FUNCTION_BLOCK FB_StateMaint
VAR_IN_OUT
	stAxis  	: ARRAY [GVL.cXP .. GVL.cXM] OF ST_AxisGroup;
	bTopEntry	: BOOL;
END_VAR
VAR_INPUT
	eCommand			: E_Commands;
	stCalibrate			: ST_Calibrate;
	stChangeAxisEnable	: ST_ChangeAxisEnable;
	stChangeBrakeState	: ST_ChangeBrakeState;
	stClearAllFaults	: ST_ClearAllFaults;
	stClearAxisFaults	: ST_ClearAxisFaults;
	stDisableAllAxes	: ST_DisableAllAxes;
	stEnableAllAxes		: ST_EnableAllAxes;
	stGoToProd			: ST_GoToProd;
	stHomeAxis			: ST_HomeAxis;
	stMoveAxisAbsolute	: ST_MoveAxisAbsolute;
	stMoveAxisRelative	: ST_MoveAxisRelative;
END_VAR
VAR_OUTPUT
	bCalibDone		: BOOL;
	bMotionDone		: BOOL;
	stOutCalibDone	: ST_CalibDone;
	nSMState		: DINT;
END_VAR
VAR
	//state-machine
	eCurrentState	: E_StatesMaint;
	eNextState		: E_StatesMaint;
	fbHoming		: FB_Homing;
	fbCalibrating	: FB_StateCalibrating;
	fbMoving		: FB_StateMoving;
	fbStill			: FB_StateStill;
	bLowerEntry 	: BOOL;

	//other var
	eCopyCommand	: E_Commands;
	fbCalibRtrig	: R_TRIG;
	bCalibRestart : BOOL;
	
	//testVar
	a, b, c : INT;
	
END_VAR


IF bTopEntry = TRUE THEN
	bTopEntry := FALSE;
	eNextState := E_StatesMaint.Still;
END_IF	
IF eCurrentState <> eNextState THEN
	bLowerEntry := TRUE;
END_IF
eCurrentState := eNextState;
nSMState := eCurrentState;
bMotionDone := FALSE;
//State Machine
CASE eCurrentState OF
	
	E_StatesMaint.Still:
		bCalibRestart := TRUE;
		fbStill(
			stAxis				:= stAxis, 
			bTopEntry			:= bLowerEntry, 
			eCommand			:= eCommand,
			stChangeAxisEnable 	:= stChangeAxisEnable,
			stChangeBrakeState	:= stChangeBrakeState,
			stClearAllFaults	:= stClearAllFaults,
			stClearAxisFaults	:= stClearAxisFaults,
			stDisableAllAxes	:= stDisableAllAxes,
			stEnableAllAxes		:= stEnableAllAxes);
		IF eCommand <> E_Commands.noCommand THEN (*checks if there is a new command*)
			IF eCommand = E_Commands.calibrate THEN
				eNextState := E_StatesMaint.Calibrating;
			ELSIF eCommand = E_Commands.closeShutter OR_ELSE
				eCommand = E_Commands.homeAxis OR_ELSE
				eCommand = E_Commands.moveAxisAbsolute OR_ELSE
				eCommand = E_Commands.moveAxisRelative THEN
					eCopyCommand := eCommand; (*need to copy since eCommand is only valid for 1 cycle. Resets to noCommand next cycle.*)
					eNextState := E_StatesMaint.Moving;
			END_IF
		END_IF
		a := a+1;
	
	E_StatesMaint.Calibrating:
		bCalibDone := FALSE;
		fbHoming(stAxis:=stAxis, bTopEntry:=bLowerEntry);
		fbCalibRtrig(CLK:=(stAxis[GVL.cXP].axisRef.Status.Homed AND stAxis[GVL.cXM].axisRef.Status.Homed AND NOT fbHoming.bBusy));
		IF fbCalibRtrig.Q THEN
			bLowerEntry:=TRUE;
		END_IF
		fbCalibrating(stAxis:=stAxis, bTopEntry:=bLowerEntry, bCalibDone:=bCalibDone, bInterrupted:=bCalibRestart, stOutCalibDone=>stOutCalibDone);
		IF bCalibDone THEN
			eNextState := E_StatesMaint.Still;
		END_IF
		b:=b+1;
		
	E_StatesMaint.Moving:
		fbMoving(
			stAxis				:= stAxis, 
			bTopEntry			:= bLowerEntry, 
			eCommand			:= eCopyCommand,
			stMoveAxisAbsolute 	:= stMoveAxisAbsolute,
			stMoveAxisRelative	:= stMoveAxisRelative);
		IF NOT fbMoving.bBusy THEN
			eNextState := E_StatesMaint.Still;
			bMotionDone := TRUE;
		END_IF
		c:=c+1;
END_CASE

END_FUNCTION_BLOCK

(* stored: Version 1.1.0.1, ProductVersion 3.1.4022.12
   POU FB_StateMaint: Id {37b42c71-d02c-4f0b-9d4a-8f4651b67341}, SpecialFunc None *)
